// TIA Portal V17 export
// export: Created 2022-03-12T16:05:33.4586376Z, ExportSetting WithDefaults, DisplayName Totally Integrated Automation Portal, DisplayVersion V17, DisplayName TIA Portal Openness, DisplayVersion V17, DisplayName TIA Portal Version Control Interface, DisplayVersion V17, DisplayName STEP 7 Professional, DisplayVersion V17, DisplayName STEP 7 Safety, DisplayVersion V17, DisplayName WinCC Advanced / Unified PC, DisplayVersion V17
TYPE "CPG_typeParameter(String)"
// stored: IsFailsafeCompliant false
   STRUCT
      ID : DInt;   // Parameter ID - This is the arbitrary (user defined) ID value of the parameter
      "Name" : String[24];   // Parameter Name - The literal parameter name is used to describe the parameter number and its associated value (e.g. Glue Temp)
      Unit : String[5];   // Parameter Unit of Measure - The parameter unit is used to describe the unit of measure of the parameter and its associated value (e.g. DegF)
      Value : String[24];   // Parameter Value - This is the numeric or string value of the parameter (e.g. '6ES7518-4AP00-0AB0')
   END_STRUCT;
END_TYPE
